FUNCTION_BLOCK Controller
  (* Standard: 61499-2 *)
  (* Version 0.1, 2015-00-08, SYY, SYY-PC *)
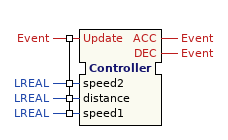
  EVENT_INPUT
    Update WITH speed2, distance, speed1;
  END_EVENT
  EVENT_OUTPUT
    ACC;
    DEC;
  END_EVENT
  VAR_INPUT
    speed2 : LREAL;
    distance : LREAL;
    speed1 : LREAL;
  END_VAR
  VAR
    sp : LREAL;
  END_VAR
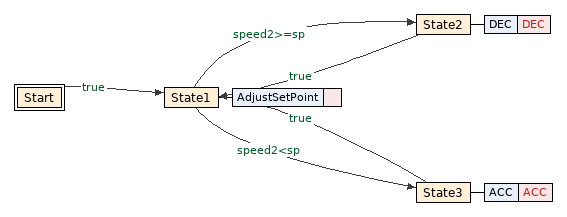
  EC_STATES
    Start;
    State1 : AdjustSetPoint;
    State2 : DEC -> DEC;
    State3 : ACC -> ACC;
  END_STATES
  EC_TRANSITIONS
    Start TO State1 := true;
    State1 TO State2 := speed2>=sp;
    State1 TO State3 := speed2<sp;
    State2 TO State1 := true;
    State3 TO State1 := true;
  END_TRANSITIONS
  ALGORITHM AdjustSetPoint IN C:
me->sp = 6.75 + 7.91 * tanh(0.13 * (me->distance - 5) - 1.57);
  END_ALGORITHM
  ALGORITHM DEC IN C:
//printf("Signal sent : the following car decelerates |  Speed1: %3.8f, Speed2: %3.8f, Distance: %3.8f\n", me->speed1, me->speed2, me->distance);
//printf("decelerate Speed1 %3.8f Speed2 %3.8f Distance %3.8f\n", me->speed1, me->speed2, me->distance);
  END_ALGORITHM
  ALGORITHM ACC IN C:
//printf("Signal sent : the following car accelerates |  Speed1: %3.8f, Speed2: %3.8f, Distance: %3.8f\n", me->speed1, me->speed2, me->distance);
//printf("accelerate Speed1 %3.8f Speed2 %3.8f Distance %3.8f\n", me->speed1, me->speed2, me->distance);
  END_ALGORITHM
END_FUNCTION_BLOCK
